// TIA Portal V20 export
DATA_BLOCK "HmiInterface"   // DB17
{ DB_Accessible_From_OPC_UA := 'FALSE' }
AUTHOR : ERsystem_FA2_DH. Kim
// stored: Access Published, DBAccessibleFromOPCUA false, DBAccessibleFromWebserver false, MemoryReserve 100, Namespace Unit1.Em0
   VAR
      em : "LAF_typeEmInterface";
      cm : Struct
         Interlock : Struct
            unwinderTopAxisB : "LER_typeAxisInterlock_Legacy";
            airShaftTopOnOff { S7_SetPoint := 'True'} : "LER_typeTwoWayActInterlock";
         END_STRUCT;
         softCam : "Unit1.type_emRelations_em0_SoftCam";
         brakeTest : Struct
            UnwinderTopAxisB : "LER_typeBrakeTestEmInterface";
         END_STRUCT;
      END_STRUCT;
      sepaUnwinderTop : Struct
         jobs { S7_SetPoint := 'True'} : "LAF_typeJobsInterface";
         sequence { S7_SetPoint := 'True'} : "LAF_typeSequenceInterface";
      END_STRUCT;
      auxiliary : Struct
         cmEpc_UnUse : Bool;
         AutoSpliceRemainingLength : LReal;
      END_STRUCT;
      cmTopDirectionCheckSensor { S7_SetPoint := 'True'} : "LBC_typeDigitalSignalInterface";
      cmRadiusMeasureTop : "LBC_typeAnalogInputInterface";
   END_VAR
   VAR RETAIN
      cmRadiusMeasure : "LER_typeRadiusMeasureInterface";
   END_VAR
   VAR
      cmUnwinderTopAxisB : "LBC_typeAxis64PosInterface";
      cmAirShaftTopOnOff : "LBC_typeTwoWayActuatorInterface";
      cmEpcTop : "LER_typeCON600Interface";
      intCondition : Struct
         Axis_01 : "LER.typeAxisIntlockAll";   // UnwinderTopAxisB
         Actuator_01 { S7_SetPoint := 'True'} : "LER.typeAxisActuatorCondition";   // UnwinderAirShaftTop
      END_STRUCT;
      motion : Struct
         jobs { S7_SetPoint := 'True'} : "LAF_typeJobsInterface";
         sequence { S7_SetPoint := 'True'} : "LAF_typeSequenceInterface";
      END_STRUCT;
      "step" : Struct
         jobs { S7_SetPoint := 'True'} : "LAF_typeJobsInterface";
         sequence { S7_SetPoint := 'True'} : "LAF_typeSequenceInterface";
      END_STRUCT;
   END_VAR
BEGIN
   cmUnwinderTopAxisB.configuration.referenceDesignator := WSTRING#'UnwinderTopAxisB';
END_DATA_BLOCK
